// TIA Portal V20 export
TYPE "UserDiag_typePLC"
TITLE = UserDiag_typePLC
   STRUCT
      hardwareId { ExternalAccessible := 'False'; ExternalVisible := 'False'; ExternalWritable := 'False'} : HW_DEVICE := 16#0000;   // Hardware identifier of the PLC
      error { ExternalAccessible := 'False'; ExternalVisible := 'False'; ExternalWritable := 'False'} : Bool := FALSE;   // TRUE: Error in PLC
      errorLedActive { ExternalAccessible := 'False'; ExternalVisible := 'False'; ExternalWritable := 'False'} : Bool := FALSE;   // TRUE: PLC led signals an error
      actualConfiguredSlots { ExternalAccessible := 'False'; ExternalVisible := 'False'; ExternalWritable := 'False'} : Int := 0;   // Number of configured local slots at PLC
      slots { ExternalAccessible := 'False'; ExternalVisible := 'False'; ExternalWritable := 'False'; S7_SetPoint := 'True'} : Array[0.."USERDIAG_SLOTS_PER_PLC_UPPER_LIM"] of "UserDiag_typeSlot";   // Information of the PLC slots; index = slotnumber; PLC always at slot 1
   END_STRUCT;
END_TYPE
